{attribute 'no_explicit_call':= 'do not call this POU directly'}
FUNCTION_BLOCK T_Monitor_Structure
VAR
    _Changed   : BOOL;
    Stored_CRC : WORD := 16#FFFF;
END_VAR

PROPERTY Changed : BOOL
GET
Changed := _Changed;
END_GET
END_PROPERTY

METHOD CyclicUpdate : BOOL
VAR_INPUT
    StructureAddress : PVOID;
	StructureLength  : UDINT;
END_VAR
VAR
    CRC : WORD;
END_VAR
CRC := F_DATA_TO_CRC16_CCITT(pData  := StructureAddress,
                             cbData := StructureLength,
                             crc    := 0);
_Changed := (CRC <> Stored_CRC);
IF Changed THEN
    Stored_CRC := CRC;
END_IF
CyclicUpdate := _Changed;
END_METHOD

METHOD Reset
VAR_INPUT
END_VAR
Stored_CRC := 16#FFFF;
_Changed   := FALSE;
END_METHOD

END_FUNCTION_BLOCK

(* stored: Version 1.1.0.1, ProductVersion 3.1.4024.12
   POU T_Monitor_Structure: Id {e37b38e2-2e88-4dba-b983-57dfb99bc7d0}, SpecialFunc None
   Folder Methods: Id {2812855e-7e80-4a08-af6c-27cc6924d195}
   Folder Properties: Id {ccfb09e6-7a9f-48ea-8a89-8d786e3554e9}
   Property Changed: Id {915cb05b-d037-4ba7-937e-8a39b6596974}
   Get Get: Id {30cd72d8-6533-4538-aa6b-cc2c5e538978}
   Method CyclicUpdate: Id {2b6fb421-e17f-4f70-ac9f-421b9e940ca2}
   Method Reset: Id {05ecd9bb-696c-41c1-98ff-be522cbd4e63} *)
